{attribute addProperty BoxType "AT2026-0250-0024"}
{attribute addProperty Id "A_0080_AT2002_5249_0019_AT2002_5249AT2002_C5E5984862678.25"}
{attribute addProperty CRC "3206552997"}
{attribute addProperty SizeInBites "626"}
{attribute addProperty SizeInBytes "78.25"}
TYPE A_0068_AT2026_0250_0024_AT2026_0250_BF201DA5 EXTENDS AT2026_BA5A9548 :
STRUCT
	{attribute addProperty Name "A_0080_AT2002_5249_0019_AT2002_5249"}
	A_0080_AT2002_5249_0019_AT2002_5249 : AT2002_C5E59848;
END_STRUCT
END_TYPE

(* stored: Version 1.2.0.0, ProductVersion 3.1.4024.9
   DUT A_0068_AT2026_0250_0024_AT2026_0250_BF201DA5: Id {5f4bea21-0c1d-4750-aa7e-eaaeafc51556} *)
